FUNCTION_BLOCK FB_Stan_Undefined EXTENDS FB_SITP_Element
VAR

END_VAR

METHOD FB_init : BOOL
VAR_INPUT
	bInitRetains : BOOL; // if TRUE, the retain variables are initialized (warm start / cold start)
	bInCopyCode : BOOL;  // if TRUE, the instance afterwards gets moved into the copy code (online change)
END_VAR
THIS^.PrzypiszTekstDo (refstEtykieta := THIS^.stNazwa, eJezyk := B_Baza.E_Jezyki.pl, wsTekst	:= "Nieokreślony");
THIS^.PrzypiszTekstDo (refstEtykieta := THIS^.stNazwa, eJezyk := B_Baza.E_Jezyki.en, wsTekst	:= "Undefined");      
THIS^.PrzypiszTekstDo (refstEtykieta := THIS^.stNazwa, eJezyk := B_Baza.E_Jezyki.de, wsTekst	:= "Nicht definiert");
END_METHOD

METHOD PUBLIC WywolajAkcjePBDlaStanu : BOOL
VAR_INPUT
	iNumerPB				: INT;
END_VAR
WywolajAkcjePBDlaStanu			:= THIS^.refstDaneSITP.refarrPB [iNumerPB].SP_Undefined ();
END_METHOD

(*			
	EVERDE sp. z o.o.
	Rafał Osajda		18.06.2025		TC 4024.66
	Zwraca true jak wyjście ze stanu jest możliwe
*)
METHOD PUBLIC ZwrocCzyMoznaWyjscZeStanu : BOOL
//warunki wyjść dla każdego ze stanów osobnym FB
IF (THIS^.refstDaneSITP.ePolecenieZmianyStanu = E_SITP_PolecenieZmianyStanu.Abort) THEN
	IF (THIS^.refstDaneSITP.arrStanyWlaczoneWTrybie [B_Baza.E_StanyPracy.Aborting]) THEN
		ZwrocCzyMoznaWyjscZeStanu					:= THIS^.ZgodaNaZmianeStanu (B_Baza.E_StanyPracy.Aborting);
	ELSE
		ZwrocCzyMoznaWyjscZeStanu					:= THIS^.BrakZgodyNaZmieneStanu (2);	//Stan do którego chcemy przejść jest wylaczony
	END_IF
ELSE
	ZwrocCzyMoznaWyjscZeStanu						:= THIS^.BrakZgodyNaZmieneStanu (1);	//Bledny rozkaz dla zmiany stanu
END_IF
END_METHOD

END_FUNCTION_BLOCK

(* stored: Version 1.1.0.1
   POU FB_Stan_Undefined: Id {01e2d724-1fbe-0ea6-02a6-b9e07ca83c1f}, SpecialFunc None
   Method FB_init: Id {254f9301-af21-06cb-3945-77e1cad64126}
   Method WywolajAkcjePBDlaStanu: Id {6e631fa3-f765-0a82-14cc-20c4d2154464}
   Method ZwrocCzyMoznaWyjscZeStanu: Id {34dae082-0745-0d04-2ab6-3337743fd6e8} *)
